{attribute 'GeneratedUsingTerminal: ELX9410-0000-0018'}
{attribute addProperty BoxType "ELX9410-0000-0018"}
{attribute addProperty Id "UndervoltageAT %I*BOOL1"}
{attribute addProperty CRC "2984778146"}
{attribute addProperty Size "1"}
TYPE Status_Us_In_B1E819A2 EXTENDS InputBase_8311D824 :
STRUCT
	{attribute addProperty Name "Undervoltage"}
	Undervoltage AT %I* : BOOL;
END_STRUCT
END_TYPE

(* stored: Version 1.2.0.0, ProductVersion 3.1.4024.9
   DUT Status_Us_In_B1E819A2: Id {b0c824dc-a21e-442e-8974-af7adb0eaa06} *)
